// SIMATIC S7-200 project (STEP 7-Micro/WIN), CPU 222 REL 02.01

ORGANIZATION_BLOCK MAIN:OB1
TITLE=PROGRAM COMMENTS
BEGIN
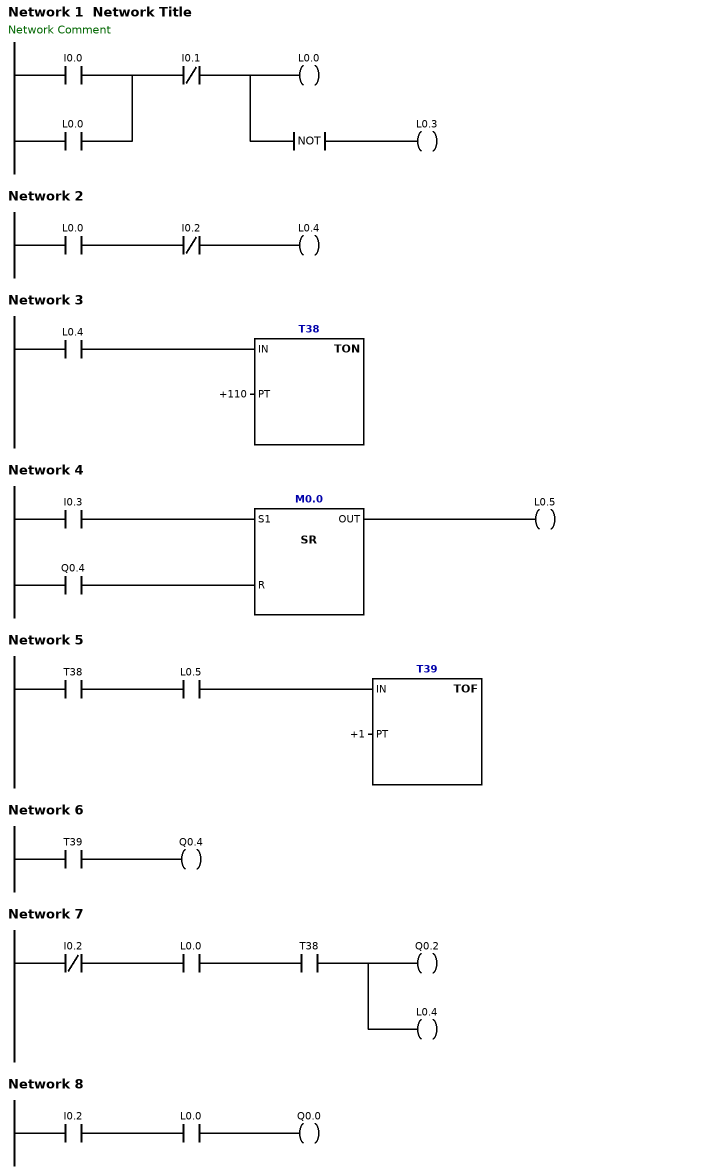
Network 1 // Network Title
// Network Comment
LD     I0.0
O      L0.0
AN     I0.1
=      L0.0
NOT
=      L0.3
Network 2
LD     L0.0
AN     I0.2
=      L0.4
Network 3
LD     L0.4
TON    T38, +110
Network 4
LD     I0.3
LD     Q0.4
NOT
A      M0.0
OLD
=      M0.0
=      L0.5
Network 5
LD     T38
A      L0.5
TOF    T39, +1
Network 6
LD     T39
=      Q0.4
Network 7
LDN    I0.2
A      L0.0
A      T38
=      Q0.2
=      L0.4
Network 8
LD     I0.2
A      L0.0
=      Q0.0
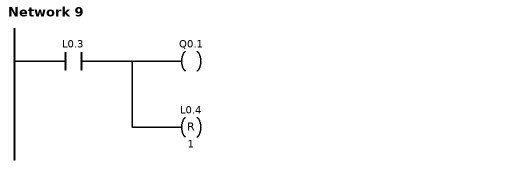
Network 9
LD     L0.3
=      Q0.1
R      L0.4, 1
END_ORGANIZATION_BLOCK
